INTERFACE I_Skill_Greifer

METHOD M_Reset : BOOL
VAR_INPUT
END_VAR
END_METHOD

METHOD M_Start : BOOL
VAR_INPUT
END_VAR
END_METHOD

METHOD M_Stop : BOOL
VAR_INPUT
END_VAR
END_METHOD

PROPERTY P_Prozessparameter : sSmartGreiferProzessVariablen
SET
END_SET
END_PROPERTY

PROPERTY P_State : eSkillState
GET
END_GET
END_PROPERTY

END_INTERFACE

(* stored: Version 1.1.0.1
   Itf I_Skill_Greifer: Id {a145d5ee-75a3-4c6d-8b40-fc175d64ee97}
   Method M_Reset: Id {6263450a-2240-4b7b-b892-40b13a134491}
   Method M_Start: Id {5541b6b8-02e8-4acd-bbd2-5599b71551a0}
   Method M_Stop: Id {94a6e96f-5049-468c-a874-8ecfa53bb572}
   Property P_Prozessparameter: Id {65b271c1-595a-42e6-adc5-106d1fc47ab6}
   Set Set: Id {c788fdea-0cfc-4503-aced-59db15aac19e}
   Property P_State: Id {35c4738c-9146-4478-8634-9a6225028fc4}
   Get Get: Id {983d46b0-cc47-4b01-8795-a39d24cbf473} *)
